(* PLC project SafeLOGIC-1, BrAutomation SafeDESIGNER  4.3.4.4 *)
(* stored: companyURL http://www.br-automation.com, creationDateTime Thu Dec 17 17:05:05 2020 *)

PROGRAM Main
  VAR  (* added by the conversion: wires and edge detectors of the diagram *)
    _OR_S29_OUT : ANY;
    _OR_S68_OUT : ANY;
    _OR_S96_OUT : ANY;
    _OR_S127_OUT : ANY;
  END_VAR

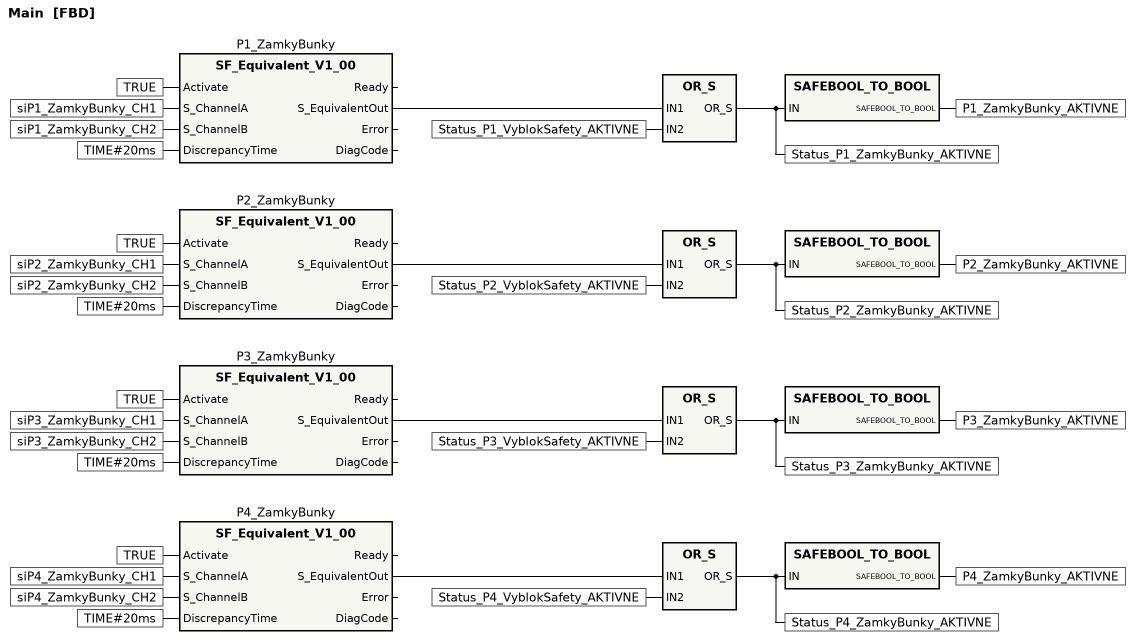
(* FBD diagram, written out as Structured Text *)
P1_ZamkyBunky(Activate := TRUE, S_ChannelA := siP1_ZamkyBunky_CH1, S_ChannelB := siP1_ZamkyBunky_CH2, DiscrepancyTime := TIME#20ms);
_OR_S29_OUT := OR_S(P1_ZamkyBunky.S_EquivalentOut, Status_P1_VyblokSafety_AKTIVNE);
Status_P1_ZamkyBunky_AKTIVNE := _OR_S29_OUT;
P1_ZamkyBunky_AKTIVNE := SAFEBOOL_TO_BOOL(_OR_S29_OUT);
P2_ZamkyBunky(Activate := TRUE, S_ChannelA := siP2_ZamkyBunky_CH1, S_ChannelB := siP2_ZamkyBunky_CH2, DiscrepancyTime := TIME#20ms);
_OR_S68_OUT := OR_S(P2_ZamkyBunky.S_EquivalentOut, Status_P2_VyblokSafety_AKTIVNE);
Status_P2_ZamkyBunky_AKTIVNE := _OR_S68_OUT;
P2_ZamkyBunky_AKTIVNE := SAFEBOOL_TO_BOOL(_OR_S68_OUT);
P3_ZamkyBunky(Activate := TRUE, S_ChannelA := siP3_ZamkyBunky_CH1, S_ChannelB := siP3_ZamkyBunky_CH2, DiscrepancyTime := TIME#20ms);
_OR_S96_OUT := OR_S(P3_ZamkyBunky.S_EquivalentOut, Status_P3_VyblokSafety_AKTIVNE);
Status_P3_ZamkyBunky_AKTIVNE := _OR_S96_OUT;
P3_ZamkyBunky_AKTIVNE := SAFEBOOL_TO_BOOL(_OR_S96_OUT);
P4_ZamkyBunky(Activate := TRUE, S_ChannelA := siP4_ZamkyBunky_CH1, S_ChannelB := siP4_ZamkyBunky_CH2, DiscrepancyTime := TIME#20ms);
_OR_S127_OUT := OR_S(P4_ZamkyBunky.S_EquivalentOut, Status_P4_VyblokSafety_AKTIVNE);
Status_P4_ZamkyBunky_AKTIVNE := _OR_S127_OUT;
P4_ZamkyBunky_AKTIVNE := SAFEBOOL_TO_BOOL(_OR_S127_OUT);
END_PROGRAM
